FUNCTION TryConvert_UINT_TO_STRING : BOOL
VAR_INPUT
	in : UINT;
	out : REFERENCE TO STRING;
END_VAR

out := UINT_TO_STRING(in);
TryConvert_UINT_TO_STRING := TRUE;

END_FUNCTION

(* stored: Version 1.1.0.1, ProductVersion 3.1.4024.12
   POU TryConvert_UINT_TO_STRING: Id {1dc1e0d6-4596-4945-84e4-8c2fad31e6c3}, SpecialFunc None *)
